PROGRAM POU
VAR
	
	i : INT := 0;
	f : REAL := 0.0;
	elapsed : TIME := TIME#0M0S0MS;
	today : DATE := DATE#2020-01-01;
	message : STRING := '';
	count : BYTE := 0;
	
	A AT %I* : BOOL := FALSE;
	B AT %I* : BOOL := FALSE;
	C AT %I* : BOOL := FALSE;
	D AT %Q* : BOOL := FALSE;
		
	op1 : INT := 1;
	op2 : INT := 2;
	res : REAL := 0.0;
	test : BOOL := FALSE;
	
	
	
	TON_0: TON;
END_VAR

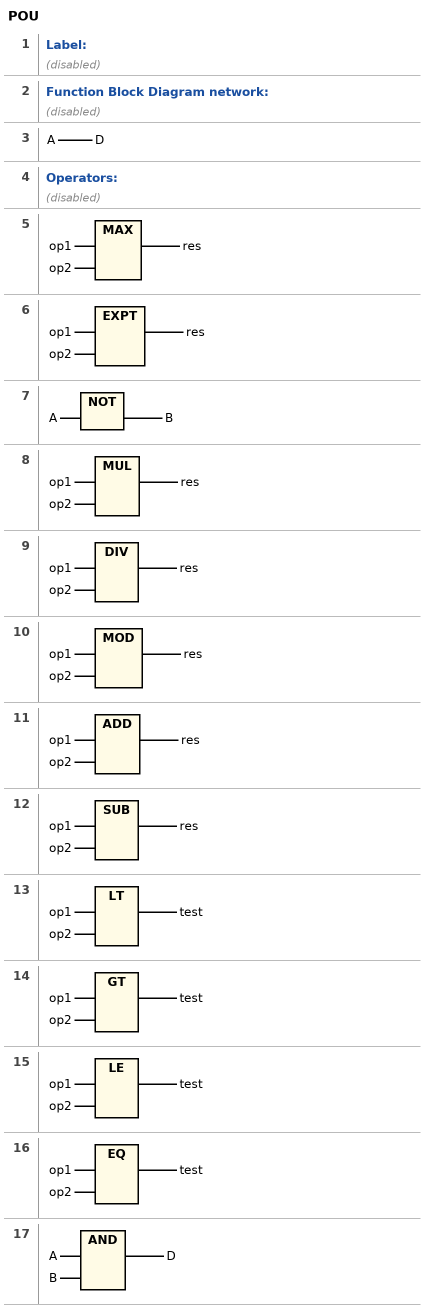
// NETWORK 1 (disabled)
// label: Label

// NETWORK 2 (disabled)
// label: Function Block Diagram network

// NETWORK 3
D := A;

// NETWORK 4 (disabled)
// label: Operators

// NETWORK 5
res := MAX(op1, op2);

// NETWORK 6
res := EXPT(op1, op2);

// NETWORK 7
B := NOT A;

// NETWORK 8
res := op1 * op2;

// NETWORK 9
res := op1 / op2;

// NETWORK 10
res := op1 MOD op2;

// NETWORK 11
res := op1 + op2;

// NETWORK 12
res := op1 - op2;

// NETWORK 13
test := op1 < op2;

// NETWORK 14
test := op1 > op2;

// NETWORK 15
test := op1 <= op2;

// NETWORK 16
test := op1 = op2;

// NETWORK 17
D := A AND B;

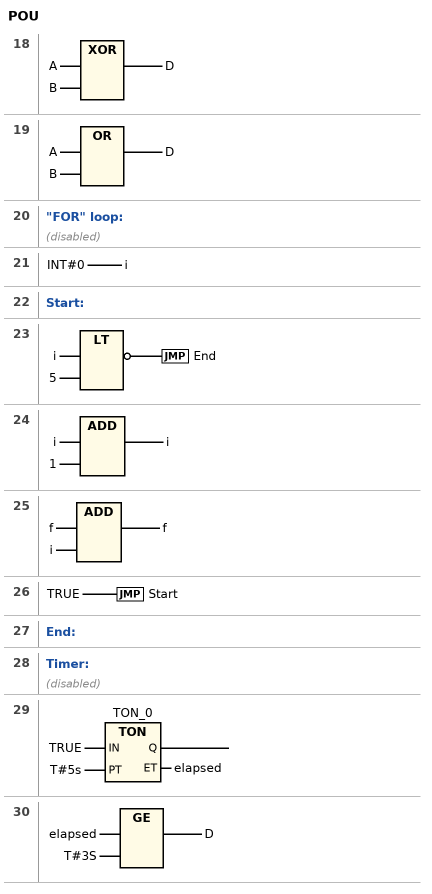
// NETWORK 18
D := A XOR B;

// NETWORK 19
D := A OR B;

// NETWORK 20 (disabled)
// label: "FOR" loop

// NETWORK 21
i := INT#0;

// NETWORK 22
Start: ;

// NETWORK 23
IF NOT (i < 5) THEN JMP End; END_IF

// NETWORK 24
i := i + 1;

// NETWORK 25
f := f + i;

// NETWORK 26
JMP Start;

// NETWORK 27
End: ;

// NETWORK 28 (disabled)
// label: Timer

// NETWORK 29
TON_0(IN := TRUE, PT := T#5s, ET => elapsed); // TON

// NETWORK 30
D := elapsed >= T#3S;

END_PROGRAM

(* stored: Version 1.1.0.1, ProductVersion 3.1.4024.3
   POU POU: Id {b221216c-99f2-4d7c-94ca-4d65839ae11c}, SpecialFunc None *)
